FUNCTION_BLOCK SSC_TransferWorkpieceTo_RampEnd EXTENDS SSC_MoveWorkpiece_Base
VAR_INPUT
END_VAR
VAR_OUTPUT
END_VAR
VAR
	// (EProcessVariables.PicAlpha_AtPos3 = TRUE) AND ((EProcessVariables.PicAlpha_HoldingWorkpiece = FALSE) AND (EProcessVariables.PicAlpha_CylinderExtended = FALSE))
	m_compExpr233: ComparisonExpression(EProcessVariables.PicAlpha_AtPos3, EComparisonType.equals, EDataType.binary, TRUE, 0, '', TRUE);
	m_compExpr235: ComparisonExpression(EProcessVariables.PicAlpha_HoldingWorkpiece, EComparisonType.equals, EDataType.binary, FALSE, 0, '', TRUE);
	m_compExpr237: ComparisonExpression(EProcessVariables.PicAlpha_CylinderExtended, EComparisonType.equals, EDataType.binary, FALSE, 0, '', TRUE);
	m_boolExpr238: BoolExpression(m_compExpr235, EBoolOperation.and_op, m_compExpr237);
	m_precondition: BoolExpression(m_compExpr233, EBoolOperation.and_op, m_boolExpr238);
	
	// TRUE
	m_postcondition: ValueExpression(EDataType.binary, TRUE, 0, '', TRUE);
	
	m_timer: TON;
	m_passby : BOOL;
END_VAR

SUPER^();

METHOD PROTECTED  AtTarget : BOOL
VAR_INPUT
END_VAR

IF m_ptrSSC^.WPAtRampEnd THEN
	m_passby := TRUE;
END_IF

IF m_passby THEN
	m_timer(IN := TRUE, PT := T#200MS);
	IF m_timer.Q THEN
		m_timer(IN := FALSE);
		m_passby := FALSE;
		AtTarget := TRUE;
	END_IF
END_IF
END_METHOD

METHOD FB_init : BOOL
VAR_INPUT
	bInitRetains : BOOL; // if TRUE, the retain variables are initialized (warm start / cold start)
	bInCopyCode : BOOL;  // if TRUE, the instance afterwards gets moved into the copy code (online change)
	
	i_ptrSSC: POINTER TO SmallSortingConveyor;
END_VAR
m_ptrSSC := i_ptrSSC;

m_id := EPrimitives.SSC_TransferWorkpieceTo_RampEnd;
m_timeout := T#200S;

Precondition := m_precondition;
Postcondition := m_postcondition;
END_METHOD

END_FUNCTION_BLOCK

(* stored: Version 1.1.0.1, ProductVersion 3.1.4024.9
   POU SSC_TransferWorkpieceTo_RampEnd: Id {fbf84c80-d5d4-46ea-a36d-5c96cb35367e}, SpecialFunc None
   Method AtTarget: Id {e7cb2f38-7e10-435e-8b4d-018f48d6f24a}
   Method FB_init: Id {9b44b6af-abaf-4bad-ad28-e1e64921cd01} *)
